// TIA Portal V17 export
// export: Created 2025-03-05T08:01:00.7341366Z, ExportSetting WithDefaults, DisplayName Totally Integrated Automation Portal, DisplayVersion V17 Update 8, DisplayName TIA Portal Openness, DisplayVersion V17 Update 8, DisplayName TIA Portal Version Control Interface, DisplayVersion V17, DisplayName SINAMICS Startdrive Advanced, DisplayVersion V17 SP2, DisplayName SINAMICS Startdrive G110M, G120, G120C, G120D, G120P, G115D, DisplayVersion V17 SP2, DisplayName SINAMICS Startdrive G130, G150, S120, S150, SINAMICS MV, S210, DisplayVersion V17 SP2, DisplayName STEP 7 Professional, DisplayVersion V17 Update 8, DisplayName SINUMERIK ONE STEP 7 Toolbox, DisplayVersion V17 Update 12, DisplayName SINUMERIK 840D sl STEP 7 Toolbox, DisplayVersion V17 Update 12, DisplayName STEP 7 Safety, DisplayVersion V17 Update 6, DisplayName WinCC Advanced, DisplayVersion V17 Update 8
DATA_BLOCK "LTLP_DeviceDiagnosticAlarmDB"   // DB597
{ DB_Accessible_From_OPC_UA := 'FALSE' }
// stored: AutoNumber true, DBAccessibleFromOPCUA false, DBAccessibleFromWebserver true, InstanceOfName LTLP_DeviceDiagnosticAlarm, InstanceOfType FB
"LTLP_DeviceDiagnosticAlarm"
   // VAR_INPUT
   //    RESTART_PLC : Bool;
   // END_VAR
   // VAR_IN_OUT
   //    HMI_DB : "LTLP_typeHmiProInterface";
   // END_VAR
   // VAR
   //    dataCounterRet : Byte;
   //    retValue : Int;
   //    HMIInterface : Struct
   //       dataCounter : Byte;
   //       systemId : Byte;
   //       stationNumber : Int;
   //       state : Byte;
   //       res : Byte;
   //    END_STRUCT;
   //    siTopStartInformation { S7_SetPoint := 'True'} : SI_classic;
   //    siStartUpClassic { S7_SetPoint := 'True'} : SI_classic;
   // END_VAR
BEGIN
END_DATA_BLOCK
